{attribute 'TcGenerated'}
// This function has been automatically generated from the project information.
VAR_GLOBAL CONSTANT
    {attribute 'const_non_replaced'}
    {attribute 'linkalways'}
    stLibVersion_lcls_plc_lfe_motion : ST_LibVersion := (iMajor := 1, iMinor := 4, iBuild := 3, iRevision := 0, sVersion := '1.4.3');
END_VAR

(* stored: Version 1.1.0.1, ProductVersion 3.1.4022.18
   GVL Global_Version: Id 51e08601-2768-49b2-b386-16600a3f7066 *)
